TYPE ST_KBUS_AnalogueDataIn :
STRUCT
	nState	: BYTE;
	nData	: INT;
END_STRUCT
END_TYPE

(* stored: Version 1.1.0.1, ProductVersion 3.1.4024.15
   DUT ST_KBUS_AnalogueDataIn: Id {b9c7adf8-4a1b-43f4-ae88-188c151027ae} *)
